FUNCTION_BLOCK FB_Counter
VAR_INPUT
	CTU	:BOOL;		// Eingang zum hoch zählen
	CTD	:BOOL;		// Eingang zum abwärts zählen
	Step:INT := 1;		// Schrittweite
END_VAR
VAR_IN_OUT
	Value: DINT;	// Zählwert
END_VAR
VAR // added by the converter: edge detectors and wires of the graphical bodies
    _rt1, _rt2 : R_TRIG;
END_VAR

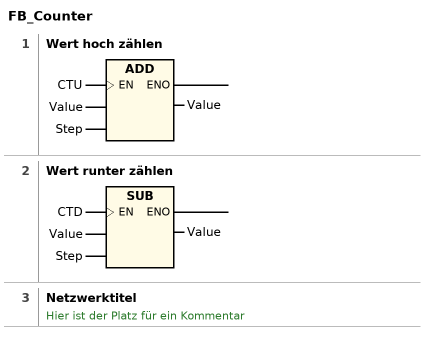
// NETWORK 1: Wert hoch zählen
_rt1(CLK := CTU);
IF _rt1.Q THEN Value := Value + Step; END_IF

// NETWORK 2: Wert runter zählen
_rt2(CLK := CTD);
IF _rt2.Q THEN Value := Value - Step; END_IF

// NETWORK 3: Netzwerktitel
// Hier ist der Platz für ein Kommentar

END_FUNCTION_BLOCK

(* stored: Version 1.1.0.1, ProductVersion 3.1.4024.12
   POU FB_Counter: Id {a71fe086-3981-4735-aa25-53c42a90aa21}, SpecialFunc None *)
